// TIA Portal project "PLC_LAB_PROCESS_AUTOMATION_SYSTEMS" (V17)

(* hardware
DEVICE "HMI_1"  KTP700 Basic PN
   slot 0: "HMI_1"  KTP700 Basic PN  6AV2 123-2GB03-0AX0  17.0.0.0
   slot 1: "HMI_RT_1"  KTP700 Basic PN  6AV2 123-2GB03-0AX0  17.0.0.0
   slot 5: "HMI_1.IE_CP_1"  PROFINET Interface  17.0.0.0
      slot 1: "PROFINET Interface_1"  PROFINET Interface
         slot 1: "Port_1"  Port
DEVICE "S7-1200 station_1"  S7-1200 Station
   slot 0: "Rack_0"  S7-1200 Rack  Rack  V1.0
   slot 1: "PLC_1"  CPU 1214C DC/DC/DC  6ES7 214-1AG40-0XB0  V4.5
*)

// ===== PLC "PLC_1"  CPU 1214C DC/DC/DC =====

VAR_GLOBAL   // PLC tag table "Default tag table"
   "START" AT %M0.0 : Bool;
   "STOP" AT %M0.1 : Bool;
   "MANUAL" AT %M0.2 : Bool;
   "AUTOMATIC" AT %M0.3 : Bool;
   "RESET_COUNTER" AT %M0.6 : Bool;
   "MOTOR" AT %MW2 : Int;
   "SENSOR_BOTTLE" AT %M1.0 : Bool;
   "status_counter" AT %MW1 : Int;
   "POWER_MEM" AT %M100.0 : Bool;
   "NEW_BOX" AT %M100.1 : Bool;
   "Clock_Byte" AT %MB200 : Byte;
   "Clock_10Hz" AT %M200.0 : Bool;
   "Clock_5Hz" AT %M200.1 : Bool;
   "Clock_2.5Hz" AT %M200.2 : Bool;
   "Clock_2Hz" AT %M200.3 : Bool;
   "Clock_1.25Hz" AT %M200.4 : Bool;
   "Clock_1Hz" AT %M200.5 : Bool;
   "Clock_0.625Hz" AT %M200.6 : Bool;
   "Clock_0.5Hz" AT %M200.7 : Bool;
END_VAR

DATA_BLOCK "conveyer_DB"   // DB2
{ S7_Optimized_Access := 'TRUE' }
VERSION : 0.1
   VAR
      reset_counter : Bool;
   END_VAR
BEGIN
END_DATA_BLOCK

// folder: System blocks/Program resources

DATA_BLOCK "BOTTLE_COUNTER"   // DB1
{ S7_Optimized_Access := 'TRUE' }
AUTHOR : Simatic
FAMILY : IEC
NAME : CNTR
VERSION : 1.0
// stored: InstanceOfName IEC_COUNTER
"IEC_COUNTER"
BEGIN
END_DATA_BLOCK

DATA_BLOCK "CONVEYER_STEPS"   // DB3
{ S7_Optimized_Access := 'TRUE' }
AUTHOR : Simatic
FAMILY : IEC
NAME : CNTR
VERSION : 1.0
// stored: InstanceOfName IEC_COUNTER
"IEC_COUNTER"
BEGIN
END_DATA_BLOCK

DATA_BLOCK "DELAY_NEXT_BOTTLE"   // DB4
{ S7_Optimized_Access := 'TRUE' }
AUTHOR : Simatic
FAMILY : IEC
NAME : IEC_TMR
VERSION : 1.0
// stored: InstanceOfName IEC_TIMER
"IEC_TIMER"
BEGIN
END_DATA_BLOCK

// folder: (top level)

ORGANIZATION_BLOCK "Main"   // OB1, LAD, ProgramCycle
TITLE = "Main Program Sweep (Cycle)"
{ S7_Optimized_Access := 'TRUE' }
VERSION : 0.1
   VAR_INPUT
      Initial_Call : Bool;   // Initial call of this OB
      Remanence : Bool;   // =True, if remanent data are available
   END_VAR
BEGIN

REGION Network 1
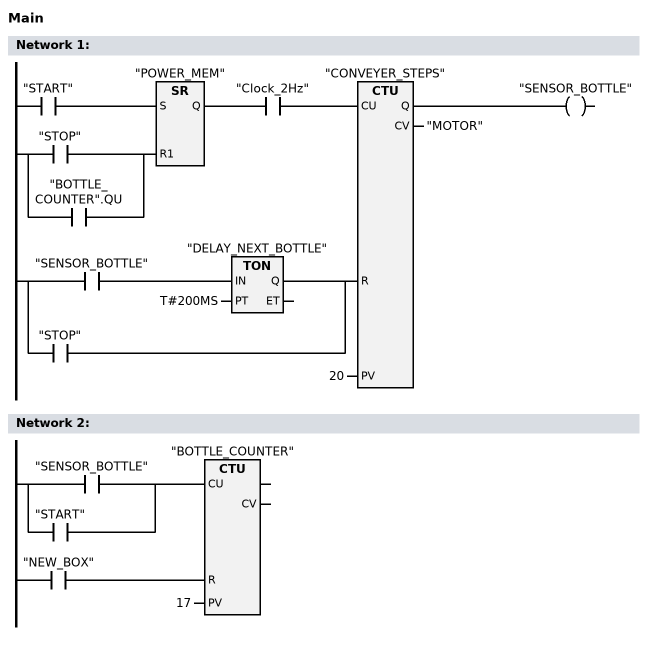
   IF "START" THEN
       "POWER_MEM" := TRUE;   // SR flip-flop
   END_IF;
   IF "STOP" OR "BOTTLE_COUNTER".QU THEN "POWER_MEM" := FALSE; END_IF;
   "DELAY_NEXT_BOTTLE".TON(IN := "SENSOR_BOTTLE", PT := T#200MS);
   "CONVEYER_STEPS".CTU(CU := "POWER_MEM" AND "Clock_2Hz",
                        R := "DELAY_NEXT_BOTTLE".Q OR "STOP",
                        PV := 20,
                        CV => "MOTOR");
   "SENSOR_BOTTLE" := "CONVEYER_STEPS".Q;
END_REGION

REGION Network 2
   "BOTTLE_COUNTER".CTU(CU := "SENSOR_BOTTLE" OR "START", R := "NEW_BOX", PV := 17);
END_REGION
END_ORGANIZATION_BLOCK

(* ===== HMI "HMI_RT_1" =====
system functions are stored by id; their names below are inferred from use
connection "HMI_Connection_1": ETHERNET, SMART_S7_1200_OMS

HMI tags "Default tag table"
   "MOTOR" : Int = PLC MOTOR AT %MW2, 1 s
   "NEW_BOX" : Bool = PLC NEW_BOX AT %M100.1, 1 s
   "START" : Bool = PLC START AT %M0.0, 1 s
   "STOP" : Bool = PLC STOP AT %M0.1, 1 s
   "MANUAL" : Bool = PLC MANUAL AT %M0.2, 1 s
   "AUTOMATIC" : Bool = PLC AUTOMATIC AT %M0.3, 1 s
   "conveyer_DB_reset_counter" : Bool = PLC conveyer_DB.reset_counter, 1 s
   "SENSOR_BOTTLE" : Bool = PLC SENSOR_BOTTLE AT %M1.0, 1 s
   "BOTTLE_COUNTER_CV" : Int = PLC BOTTLE_COUNTER.CV, 1 s

screen "Screen_1" 800x480
   Button "Button_1" at 25,14 size 123x46; TextOff 'Auto'
      Appearance <- "AUTOMATIC"
   Button "Button_3" at 25,74 size 123x46; TextOff 'Manual'
      Appearance <- "MANUAL"
   Button "Button_2" at 24,423 size 99x44; TextOff 'Start'
      on Press: SetBit("START")
      on Release: ResetBit("START")
   Button "Button_4" at 135,423 size 99x44; TextOff 'Stop'
      on Press: SetBit("STOP")
      on Release: ResetBit("STOP")
   GraphicView "Graphic view_1" at 13,249 size 471x82; Picture "Graphic_2"
   GraphicView "Graphic view_2" at 83,192 size 32x85; Picture "Graphic_3"
      HorizontalMovement <- "MOTOR"
   Button "Button_5" at 553,15 size 242x77; TextOff 'New Box'
      on Press: SetBit("NEW_BOX")
      on Release: ResetBit("NEW_BOX")
   Circle "Circle_1" at 740,423 size 48x48
      Visibility <- "BOTTLE_COUNTER_CV"
   Circle "Circle_2" at 669,423 size 48x48
      Visibility <- "BOTTLE_COUNTER_CV"
   Circle "Circle_3" at 601,423 size 48x48
      Visibility <- "BOTTLE_COUNTER_CV"
   Circle "Circle_4" at 532,423 size 48x48
      Visibility <- "BOTTLE_COUNTER_CV"
   Circle "Circle_5" at 532,369 size 48x48
      Visibility <- "BOTTLE_COUNTER_CV"
   Circle "Circle_6" at 532,309 size 48x48
      Visibility <- "BOTTLE_COUNTER_CV"
   Circle "Circle_7" at 532,249 size 48x48
      Visibility <- "BOTTLE_COUNTER_CV"
   Circle "Circle_8" at 601,369 size 48x48
      Visibility <- "BOTTLE_COUNTER_CV"
   Circle "Circle_9" at 601,309 size 48x48
      Visibility <- "BOTTLE_COUNTER_CV"
   Circle "Circle_10" at 601,249 size 48x48
      Visibility <- "BOTTLE_COUNTER_CV"
   Circle "Circle_11" at 669,249 size 48x48
      Visibility <- "BOTTLE_COUNTER_CV"
   Circle "Circle_12" at 737,249 size 48x48
      Visibility <- "BOTTLE_COUNTER_CV"
   Circle "Circle_13" at 669,311 size 48x48
      Visibility <- "BOTTLE_COUNTER_CV"
   Circle "Circle_14" at 740,305 size 48x48
      Visibility <- "BOTTLE_COUNTER_CV"
   Circle "Circle_15" at 669,365 size 48x48
      Visibility <- "BOTTLE_COUNTER_CV"
   Circle "Circle_16" at 740,365 size 48x48
      Visibility <- "BOTTLE_COUNTER_CV"
*)